(* Sample server application. Adapt this code to match your needs. *)
FUNCTION_BLOCK FB_ServerApplication
VAR_IN_OUT
	fbTx 			: FB_FrameFifo;(* TX fifo *)
	fbRx 			: FB_FrameFifo;(* RX fifo *)
	fbLog			: FB_LogFifo;(* Log message fifo *)
END_VAR
VAR
	stToClient		: ST_Input_Output; (* Tx user data *)
	stFromClient	: ST_Input_Output; (* Rx user data *)
	sLogMessage 	: T_MaxString := '';(* Log/debug/error message *)
	velInputControl	: LREAL := 0;
	torqPidControl: FB_BasicPID;
	resetPID		: BOOL := TRUE;
	PIDval			: LREAL := 0;
END_VAR

(*------------------- Fetch rx data and send them back to the client -------------------------------------------------- *)
REPEAT
	fbRx.RemoveHead( );(* Fetch data from rx fifo *)
	IF fbRx.bOk THEN(* Success *)
		stFromClient := fbRx.stGet;
		velInputControl := stFromClient.rpmout_speedin;
		
		(* Following PID controller is the crise control. This emulates the intelligent machine throttle/brake. *)
		(* ToDo find some reasonable PID parameters *)
		torqPidControl(
			fSetpointValue:= PLCPRJ_CRUISE_CONTROL_SET, 
			fActualValue:= velInputControl, 
			bReset:= resetPID, 
			fCtrlCycleTime:= 0.00025, 
			fKp:= 120,
			fTn:= 2, 
			fTv:= 1, 
			fTd:= 0.2);
		IF torqPidControl.fCtrlOutput >= 600 THEN
			PIDval := 600;
		ELSIF torqPidControl.fCtrlOutput <= -600 THEN
			PIDval := -600;
		ELSE
			PIDval := torqPidControl.fCtrlOutput;
		END_IF
		resetPID := FALSE;
		(* Set the got and calculated values. First to servos and then to Mevea *)
		(* Velocity is the angular velocity of the motor. Should be scaled possibly *)
		SetVelocity :=REAL_TO_INT(velInputControl);
		(* Max torque is set to +-600. Can be adjusted from mevea *)
		SetTorque := REAL_TO_INT(PIDval);
		
		stToClient.brake :=0;
		stToClient.rpmin_torqout :=PIDval;
		stToClient.rpmout_speedin :=1;

		(* Send data back to the client *)
		fbTx.AddTail( stPut := stToClient );(* Put user data to the tx fifo *)
		IF NOT fbTx.bOk THEN(* Fifo overflow => Log error *)
			fbLog.Error( sMessage := 'FB_FrameFifo(sender)', nErrID := PLCPRJ_ERROR_SENDFIFO_OVERFLOW );
		END_IF
	END_IF
UNTIL NOT fbRx.bOk
END_REPEAT

(*---------------------- Get log/error messages from log fifo ------------------*)
REPEAT
	fbLog.Remove( );
	IF fbLog.bOk THEN

		(* TODO: Implement log message handler *)
		sLogMessage := fbLog.sGet;

	END_IF
UNTIL NOT fbLog.bOk
END_REPEAT

END_FUNCTION_BLOCK

(* stored: Version 1.1.0.1, ProductVersion 3.1.4024.5
   POU FB_ServerApplication: Id {27aa47e1-a593-472a-a33b-33b9fe6bd70e}, SpecialFunc None *)
